TYPE ST_P_SET_RECIPE_COND :
STRUCT
	RecipeName:					STRING;
END_STRUCT
END_TYPE

(* stored: Version 1.1.0.1, ProductVersion 3.1.4024.10
   DUT ST_P_SET_RECIPE_COND: Id {218c6841-88a6-440f-a75d-6bf978b8bc28} *)
